// TIA Portal V17 export
// export: Created 2023-03-06T02:05:26.8870824Z, ExportSetting WithDefaults, DisplayName Totally Integrated Automation Portal, DisplayVersion V17 Update 4, DisplayName TIA Portal Openness, DisplayVersion V17 Update 4, DisplayName TIA Portal Version Control Interface, DisplayVersion V17, DisplayName STEP 7 Professional, DisplayVersion V17 Update 4, DisplayName STEP 7 Safety, DisplayVersion V17, DisplayName WinCC Professional, DisplayVersion V17 Update 4
TYPE "R_MV"
// stored: IsFailsafeCompliant false
   STRUCT
      xTrafo1TempTripSt : Bool;   // U11.DI0.0
      xTrafo1TempAlmSt : Bool;   // U11.DI0.1
      xTrafo1PressTripSt : Bool;   // U11.DI0.2
      xTrafo1OilLevTripSt : Bool;   // U11.DI0.3
      xLine1DiscOpenSt : Bool;   // U11.DI0.4
      xLine1DiscCloseSt : Bool;   // U11.DI0.5
      xLine1GndCloseSt : Bool;   // U11.DI0.6
      xProt1GasPress1St : Bool;   // U11.DI0.7
      xLine2DiscOpenSt : Bool;   // U11.DI1.0
      xLine2DiscCloseSt : Bool;   // U11.DI1.1
      xLine2GndCloseSt : Bool;   // U11.DI1.2
      xProt1DiscCloseSt : Bool;   // U11.DI1.3
      xProt1DiscOpenSt : Bool;   // U11.DI1.4
      xProt1GndCloseSt : Bool;   // U11.DI1.5
      xProt1CircBrkOpenSt : Bool;   // U11.DI1.6
      xProt1CircBrkCloseSt : Bool;   // U11.DI1.7
      xProt1RelayFltSt : Bool;   // U12.DI0.0
      xLV1SurgeProtSt : Bool;   // U12.DI0.1
      xSpring1ChargeSt : Bool;   // U12.DI0.2
      xProt1GasPress2St : Bool;   // U12.DI0.3
      xBackfeedtrakers1St : Bool;   // U12.DI0.4
      xProt1NeutrSurgeFltSt : Bool;   // U12.DI0.5
      xLVS1SmokeDetecSt : Bool;   // U12.DI0.6
      xSmoke1DetecSt : Bool;   // U12.DI0.7
      xSAI1SmokeDetecSt : Bool;   // U12.DI1.0
      xSSAA1SmokeDetecSt : Bool;   // U12.DI1.1
      xAirCond1AlmSt : Bool;   // U12.DI1.2
      xAcBrkHENK1OpenSt : Bool;   // U12.DI1.3
      xAcBrkHENK1CloseSt : Bool;   // U12.DI1.4
      xTrafo2TempTripSt : Bool;   // U12.DI1.5
      xTrafo2TempAlmSt : Bool;   // U12.DI1.6
      xTrafo2PressTripSt : Bool;   // U12.DI1.7
      xTrafo2OilLevTripSt : Bool;   // U13.DI0.0
      xProt2DiscCloseSt : Bool;   // U13.DI0.1
      xProt2DiscOpenSt : Bool;   // U13.DI0.2
      xProt2GndCloseSt : Bool;   // U13.DI0.3
      xProt2CircBrkOpenSt : Bool;   // U13.DI0.4
      xProt2CircBrkCloseSt : Bool;   // U13.DI0.5
      xProt2NCWatchdogSt : Bool;   // U13.DI0.6
      xLV2SurgeProtSt : Bool;   // U13.DI0.7
      xSpring2ChargeSt : Bool;   // U13.DI1.0
      xAcBrkHENK2OpenSt : Bool;   // U13.DI1.1
      xAcBrkHENK2CloseSt : Bool;   // U13.DI1.2
      xBackfeedtrakers2St : Bool;   // U13.DI1.3
      xProt2NeutrSurgeSt : Bool;   // U13.DI1.4
      xSAI2SmokeDetecSt : Bool;   // U13.DI1.5
      xSSAA2SmokeDetecSt : Bool;   // U13.DI1.6
      xAirCond2AlmSt : Bool;   // U13.DI1.7
      rPT100Trafo1St : Real;   // U15.AI0
      rPT100Trafo2St : Real;   // U15.AI1
   END_STRUCT;
END_TYPE
